# EPICS substitutions: tjmperSup/tjmper_error_setter.substitutions
file $(UTILITIES)/db/error_setter.template {
    pattern {P, STREAM_PV, PV_NAME}

    {"\$(P)", "ID", "MODE"}
    {"\$(P)", "ID", "LMT"}
    {"\$(P)", "ID", "AIR"}
    {"\$(P)", "ID", "ERR"}
}
